INTERFACE I_Wildcards

METHOD Asterisk : I_PathGenerator
VAR_INPUT
	left	: Tc2_System.T_MaxString;
	right	: Tc2_System.T_MaxString;
END_VAR
END_METHOD

METHOD Questionmark : I_PathGenerator
VAR_INPUT
END_VAR
END_METHOD

END_INTERFACE

(* stored: Version 1.1.0.1, ProductVersion 3.1.4024.14
   Itf I_Wildcards: Id {ad4ccec5-364c-0839-382d-fc6bce9721ba}
   Method Asterisk: Id {3499261a-9b3d-0eb0-0832-99df6b3cd2b3}
   Method Questionmark: Id {3b82a598-06cc-065d-24a6-80e901df76f0} *)
